(* CODESYS project SPT_Utilities.library
   Company: Beckhoff Automation LLC
   DefaultNamespace: SPT_Utilities
   Version: 3.0.3
   Placeholder: SPT Utilities
   Title: SPT Utilities

Project tree, tasks and I/O mapping:
  libraries: SPT Base Types, * (Beckhoff Automation LLC); Tc2_System, * (Beckhoff Automation GmbH); Tc3_EventLogger, * (Beckhoff Automation GmbH); Tc3_JsonXml, * (Beckhoff Automation GmbH); Tc3_Module, * (Beckhoff Automation GmbH)
  Analog Scaling/
    DUT/
      data type ST_ScalingParameters
    function F_ApplyScaling [ST]
  Buffers/
    function block FB_FIFO_ULINT_Array [ST]: AddEntry, EntryCount, LastInValue, NextOutValue, RemoveEntry
  Helper/
    function F_CompareLREAL [ST]
    function F_CompareREAL [ST]
    function F_LREAL_RoundToPlace [ST]
    function block FB_SimpleRateLimiter [ST]
  Project Information/
    function F_GetCompany [ST]
    function F_GetTitle [ST]
    function F_GetVersion [ST]
  Trace Listener/
    function block FB_MessageListener [ST]: Listener, OnMessageSent
    function block FB_TraceListenerBase [ST]: CyclicLogic, Initialize, OnTraceReceived
    interface I_TraceListener: OnTraceReceived
    data type ST_TraceMessage
  Tree_IndexBased/
    function block FB_Tree_IndexBased [ST]: AddNodeAsChildByName, GetIndexByName, Initialize
    interface I_Tree_IndexBased: AddNodeAsChildByName
    data type ST_Tree_IndexBased_Node
  Version/
    global variables Global_Version
*)

// Analog Scaling/DUT/ST_ScalingParameters
TYPE ST_ScalingParameters :
STRUCT
	Input_Minimum : LREAL := 0;
	Input_Maximum : LREAL := 100;
	Output_Minimum : LREAL := 0;
	Output_Maximum : LREAL := 4096;
END_STRUCT
END_TYPE

// Trace Listener/ST_TraceMessage
TYPE ST_TraceMessage :
    STRUCT
        Timestamp : T_MaxString;
        Source    : T_MaxString;
        Context   : T_MaxString;
        ScanCount : UDINT;
        Flags     : UDINT;
        Message   : T_MaxString;
        Json      : T_MaxString;
    END_STRUCT
END_TYPE

// Tree_IndexBased/ST_Tree_IndexBased_Node
TYPE ST_Tree_IndexBased_Node :
    STRUCT
        Name       : STRING;
        ChildCount : DINT;
        Parent     : DINT;
        Children   : ARRAY[0..15] OF DINT;
        Depth      : DINT;
    END_STRUCT
END_TYPE

// Version/Global_Version
{attribute 'TcGenerated'}
{attribute 'no-analysis'}
{attribute 'linkalways'}
// This function has been automatically generated from the project information.
VAR_GLOBAL CONSTANT
	{attribute 'const_non_replaced'}
	stLibVersion_SPT_Utilities : ST_LibVersion := (iMajor := 3, iMinor := 0, iBuild := 3, iRevision := 0, nFlags := 1, sVersion := '3.0.3');
END_VAR

// Analog Scaling/F_ApplyScaling
FUNCTION F_ApplyScaling : LREAL
VAR_INPUT
	X : LREAL;
	Parameters : ST_ScalingParameters;
END_VAR
VAR
	Slope : LREAL;
END_VAR

IF Parameters.Input_Minimum >= Parameters.Input_Maximum THEN
	//Error -- no span to scale
	F_ApplyScaling := 0;
	RETURN;
ELSIF Parameters.Output_Minimum >= Parameters.Output_Maximum THEN
	//Error -- no span to scale
	F_ApplyScaling := 0;
	RETURN;

END_IF

//Input is pegged
IF X <= Parameters.Input_Minimum THEN
	F_ApplyScaling := Parameters.Output_Minimum;
	RETURN;
ELSIF X >= Parameters.Input_Maximum THEN
	F_ApplyScaling := Parameters.Output_Maximum;
	RETURN;
END_IF

//I/O ok--scale it
IF (Parameters.Input_Maximum - Parameters.Input_Minimum) <> 0.0 THEN
	Slope := (Parameters.Output_Maximum - Parameters.Output_Minimum) / (Parameters.Input_Maximum - Parameters.Input_Minimum);
ELSE
	Slope := 0.0;
END_IF

F_ApplyScaling := Slope * (X - Parameters.Input_Minimum) + Parameters.Output_Minimum ;

END_FUNCTION

// Buffers/FB_FIFO_ULINT_Array
//! @summary A general purpose FIFO buffer for the ULINT (64-bit Unsigned Integer) datatype
FUNCTION_BLOCK FB_FIFO_ULINT_Array
VAR_IN_OUT
    Buffer : ARRAY[*] OF ULINT;
END_VAR
VAR
    _EntryCount : DINT;
END_VAR

//! @summary Adds an entry to the buffer

METHOD AddEntry : BOOL //! TRUE if entry was accepted, FALSE if buffer is full
VAR_INPUT
    Entry : ULINT; //! Entry to add
END_VAR
VAR
    i : DINT;
END_VAR
IF (LOWER_BOUND(Buffer, 1) + _EntryCount - 1) > UPPER_BOUND(Buffer, 1) THEN
    AddEntry := FALSE; //FIFO is full
ELSE
    FOR i := UPPER_BOUND(Buffer, 1) - 1 TO LOWER_BOUND(Buffer, 1) BY -1 DO
        Buffer[i + 1] := Buffer[i];
    END_FOR

    Buffer[LOWER_BOUND(Buffer, 1)] := Entry;

    _EntryCount := _EntryCount + 1;
    AddEntry    := TRUE;
END_IF
END_METHOD

//! @summary Returns the number of entries in the buffer
PROPERTY EntryCount : DINT
GET
EntryCount := _EntryCount;
END_GET
END_PROPERTY

//! @summary Returns the last entry placed in the buffer
PROPERTY LastInValue : ULINT
GET
IF _EntryCount = 0 THEN
    LastInValue := 0;
ELSE
    LastInValue := Buffer[LOWER_BOUND(Buffer, 1)];
END_IF
END_GET
END_PROPERTY

//! @summary Returns the head entry of the buffer
PROPERTY NextOutValue : ULINT
GET
IF _EntryCount = 0 THEN
    NextOutValue := 0;
ELSE
    NextOutValue := Buffer[LOWER_BOUND(Buffer, 1) + _EntryCount - 1];
END_IF
END_GET
END_PROPERTY

//! @summary Removes head entry from the buffer

METHOD RemoveEntry : BOOL //! TRUE if entry was removed, FALSE if the buffer was already empty
VAR
    i : DINT;
END_VAR
IF _EntryCount = 0 THEN
    RemoveEntry := FALSE;
ELSE
    IF (LOWER_BOUND(Buffer, 1) + _EntryCount - 1) <= UPPER_BOUND(Buffer, 1) THEN
        Buffer[LOWER_BOUND(Buffer, 1) + _EntryCount - 1] := 0;
        _EntryCount                                      := _EntryCount - 1;
        RemoveEntry                                      := TRUE;
    END_IF
END_IF
END_METHOD

END_FUNCTION_BLOCK

// Helper/F_CompareLREAL
FUNCTION F_CompareLREAL : BOOL
VAR_INPUT
    Val1      : LREAL;
    Val2      : LREAL;
    Tolerance : LREAL;
END_VAR

F_CompareLREAL := ABS(Val1 - Val2) < Tolerance;

END_FUNCTION

// Helper/F_CompareREAL
FUNCTION F_CompareREAL : BOOL
VAR_INPUT
    Val1      : REAL;
    Val2      : REAL;
    Tolerance : REAL;
END_VAR

F_CompareREAL := ABS(Val1 - Val2) < Tolerance;

END_FUNCTION

// Helper/F_LREAL_RoundToPlace
                                      //! @summary Rounds an LREAL to a given number of decimal places
FUNCTION F_LREAL_RoundToPlace : LREAL //! Rounded number
VAR_INPUT
    In            : LREAL; //! Number to be rounded
    DecimalPlaces : DINT;  //! Number of decimal places
END_VAR
VAR
END_VAR

F_LREAL_RoundToPlace := DINT_TO_LREAL(LREAL_TO_DINT(In * (DecimalPlaces * 10))) / (DecimalPlaces * 10);

END_FUNCTION

// Helper/FB_SimpleRateLimiter
FUNCTION_BLOCK FB_SimpleRateLimiter
VAR_INPUT
	Enable		  : BOOL;
	TargetValue	  : LREAL;
	Minimum		  : LREAL;
	Maximum		  : LREAL;
	Rate_Increase : LREAL; //Units per second
	Rate_Decrease : LREAL; //Units per second
END_VAR

VAR_OUTPUT
	Y : LREAL;
END_VAR

VAR
	CycleTime_Seconds	 : LREAL;
	IncreaseRatePerCycle : LREAL;
	DecreaseRatePerCycle : LREAL;
END_VAR

IF CycleTime_Seconds = 0 THEN
	CycleTime_Seconds := UDINT_TO_LREAL(TwinCAT_SystemInfoVarList._TaskInfo[GETCURTASKINDEXEX()].CycleTime) / 10000000.0;
END_IF

IF Enable THEN
	IncreaseRatePerCycle := Rate_Increase * CycleTime_Seconds;
	DecreaseRatePerCycle := Rate_Decrease * CycleTime_Seconds;
	IF Y <> TargetValue THEN
		IF TargetValue < Y THEN
			//Decrease output
			Y := Y - DecreaseRatePerCycle;
			IF Y < Minimum THEN
				Y := Minimum;
			END_IF
		ELSIF TargetValue > Y THEN
			//Increase output
			Y := Y + IncreaseRatePerCycle;
			IF Y > Maximum THEN
				Y := Maximum;
			END_IF
		END_IF
	END_IF
END_IF

END_FUNCTION_BLOCK

// Project Information/F_GetCompany
// This function has been automatically generated from the project information.
{attribute 'signature_flag' := '1073741824'}
{attribute 'TcGenerated'}
{attribute 'no-analysis'}
FUNCTION F_GetCompany : WSTRING
VAR_INPUT
	
END_VAR

F_GetCompany := "Beckhoff Automation LLC";

END_FUNCTION

// Project Information/F_GetTitle
// This function has been automatically generated from the project information.
{attribute 'signature_flag' := '1073741824'}
{attribute 'TcGenerated'}
{attribute 'no-analysis'}
FUNCTION F_GetTitle : WSTRING
VAR_INPUT
	
END_VAR

F_GetTitle := "SPT Utilities";

END_FUNCTION

// Project Information/F_GetVersion
// This function has been automatically generated from the project information.
{attribute 'signature_flag' := '1073741824'}
{attribute 'TcGenerated'}
{attribute 'no-analysis'}
FUNCTION F_GetVersion : ST_LibVersion
VAR_INPUT
	
END_VAR

F_GetVersion.iMajor := 3;
F_GetVersion.iMinor := 0;
F_GetVersion.iBuild := 3;
F_GetVersion.iRevision := 0;
F_GetVersion.sVersion := '3.0.3';
F_GetVersion.nFlags := 1;

END_FUNCTION

// Trace Listener/FB_MessageListener
FUNCTION_BLOCK FINAL FB_MessageListener EXTENDS FB_ListenerBase2
VAR
    Json          : FB_JsonDomParser; //Parse JSON attribute of messages
    JsonAttribute : STRING(10000);    //Holds JSON attribute
    hr            : HRESULT;          //Signals JSON attribute was successfully read
    ipListener    : I_TraceListener;  //Receives callback once message is processed
END_VAR

PROPERTY Listener : I_TraceListener
SET
ipListener := Listener;
END_SET
END_PROPERTY

METHOD OnMessageSent : HRESULT
VAR_INPUT
    fbEvent : REFERENCE TO FB_TcEvent;
END_VAR

VAR
    Message      : ST_TraceMessage;
    JsonDocument : SJsonValue;
    JsonProperty : SJsonValue;
END_VAR
hr := fbEvent.GetJsonAttribute(JsonAttribute, SIZEOF(JsonAttribute));
IF SUCCEEDED(hr) THEN
    JsonDocument := Json.ParseDocument(JsonAttribute);
    IF Json.HasMember(JsonDocument, 'DCTimeStamp') THEN
        JsonProperty      := Json.FindMember(JsonDocument, 'DCTimeStamp');
        Message.Timestamp := Json.GetString(JsonProperty);
    END_IF

    IF Json.HasMember(JsonDocument, 'Instance') THEN
        JsonProperty   := Json.FindMember(JsonDocument, 'Instance');
        Message.Source := Json.GetString(JsonProperty);
    END_IF

    IF Json.HasMember(JsonDocument, 'Context') THEN
        JsonProperty    := Json.FindMember(JsonDocument, 'Context');
        Message.Context := Json.GetString(JsonProperty);
    END_IF

    IF Json.HasMember(JsonDocument, 'ScanCount') THEN
        JsonProperty      := Json.FindMember(JsonDocument, 'ScanCount');
        Message.ScanCount := Json.GetUint(JsonProperty);
    END_IF

    IF Json.HasMember(JsonDocument, 'Flags') THEN
        JsonProperty  := Json.FindMember(JsonDocument, 'Flags');
        Message.Flags := Json.GetUint(JsonProperty);
    END_IF

    IF Json.HasMember(JsonDocument, 'Message') THEN
        JsonProperty    := Json.FindMember(JsonDocument, 'Message');
        Message.Message := Json.GetString(JsonProperty);
    END_IF

    IF Json.HasMember(JsonDocument, 'ExtendedInfo') THEN
        JsonProperty := Json.FindMember(JsonDocument, 'ExtendedInfo');
        Message.Json := Json.GetString(JsonProperty);
    END_IF

    IF ipListener <> 0 THEN
        //Notify listener of message data
        ipListener.OnTraceReceived(Message);
    END_IF
END_IF

OnMessageSent := S_OK; // in order to receive more callbacks (Set <> S_OK in order to cancel the callbacks for this program cycle.)
END_METHOD

END_FUNCTION_BLOCK

// Trace Listener/I_TraceListener
INTERFACE I_TraceListener

METHOD OnTraceReceived
VAR_INPUT
    Message : ST_TraceMessage;
END_VAR
END_METHOD

END_INTERFACE

// Trace Listener/FB_TraceListenerBase
FUNCTION_BLOCK ABSTRACT FB_TraceListenerBase EXTENDS FB_CyclicFB IMPLEMENTS I_TraceListener
VAR_INPUT
END_VAR

VAR_OUTPUT
END_VAR

VAR
    MessageListener : FB_MessageListener;
END_VAR

METHOD PUBLIC CyclicLogic
IF NOT _InitComplete THEN
    _InitComplete := Initialize();
    RETURN;
END_IF

MessageListener.Execute();
END_METHOD

METHOD PROTECTED Initialize : BOOL
VAR
    ListenerFilter : FB_TcEventFilter;
    hr             : HRESULT;
END_VAR
MessageListener.Listener := THIS^;                                   //For callbacks on message received
ListenerFilter.Clear().EventClass.EqualTo(TC_EVENT_CLASSES.Tracing); //Filter events by tracing class
hr := MessageListener.Subscribe2(ListenerFilter);                    //Subscribe to retrieve defined events
IF SUCCEEDED(hr) THEN
    Initialize := TRUE;
END_IF
END_METHOD

METHOD ABSTRACT OnTraceReceived
VAR_INPUT
    Message : ST_TraceMessage;
END_VAR
//Override this method to implement your specific handling
END_METHOD

END_FUNCTION_BLOCK

// Tree_IndexBased/FB_Tree_IndexBased
//! @summary Maintains a hierachical representation of a group of parent/child relationships 
FUNCTION_BLOCK FB_Tree_IndexBased IMPLEMENTS I_Tree_IndexBased
VAR_IN_OUT
    Nodes : ARRAY[0..63] OF ST_Tree_IndexBased_Node; //! Holding array
END_VAR
VAR_INPUT
    Head : STRING; //Name of the root element
END_VAR
VAR
    Initialized  : BOOL;
    NodeCount    : DINT;
    NewNodeIndex : DINT;
    HeadIndex    : DINT;

    //"Temp" variables for use in AddNodeAsChildByName
    ParentIndex : DINT;
    ChildCount  : DINT;
END_VAR

IF NOT Initialized THEN
    Initialize();
END_IF

//! @summary Add a child element to a node
METHOD AddNodeAsChildByName
VAR_INPUT
    NewName    : STRING; //! Name of the new element
    ParentName : STRING; //! Name of the parent element
END_VAR
ParentIndex := GetIndexByName(ParentName); //Find the index value of the designated parent node
ChildCount  := Nodes[ParentIndex].ChildCount;

IF ParentIndex >= 0 THEN                                        //If GetIndex was successful
    IF (Nodes[ParentIndex].ChildCount < 64) THEN                //TODO: Proper Constant bound definition	//If the parent is not at max child count
        Nodes[NewNodeIndex].Name                := NewName;     //assign new node name to next empty node in list
        Nodes[NewNodeIndex].Parent              := ParentIndex; //assign the parent node to the new child node
        Nodes[NewNodeIndex].Depth               := Nodes[ParentIndex].Depth + 1;
        Nodes[ParentIndex].Children[ChildCount] := NewNodeIndex; //assign the new node location as the next child in the parent

        NewNodeIndex                  := NewNodeIndex + 1; //Increment to next empty node
        Nodes[ParentIndex].ChildCount := ChildCount + 1;
    END_IF
END_IF
END_METHOD

//! @summary Searches the current branch for a node matching the provided name and returns its index
//! The index of the matching node (-1 if no match found)
METHOD PUBLIC GetIndexByName : DINT
VAR_INPUT
    Name : STRING; //! Node to search for
END_VAR
VAR
    i : DINT;
END_VAR
FOR i := 0 TO NodeCount DO
    IF Nodes[i].Name = Name THEN
        GetIndexByName := i;
        RETURN;
    END_IF
END_FOR

GetIndexByName := -1;
END_METHOD

METHOD PRIVATE Initialize
NodeCount := 64;

IF NodeCount >= 0 THEN
    HeadIndex               := 0;
    Nodes[HeadIndex].Name   := Head;
    Nodes[HeadIndex].Depth  := 0;
    Nodes[HeadIndex].Parent := -1;
    NewNodeIndex            := HeadIndex + 1;
END_IF
END_METHOD

END_FUNCTION_BLOCK

// Tree_IndexBased/I_Tree_IndexBased
INTERFACE I_Tree_IndexBased

METHOD PUBLIC AddNodeAsChildByName
VAR_INPUT
    NewName    : STRING;
    ParentName : STRING;
END_VAR
END_METHOD

END_INTERFACE
